(*

.. <legal notes>

legal notes
=================
| SPDX-FileCopyrightText: © 2026 Oleksandr Tiutyk <trofimich@gmail.com>
| SPDX-License-Identifier: LGPL-3.0-only
| For details check: LGPL-3.0-only_

.. _LGPL-3.0-only: https://www.gnu.org/licenses/lgpl-3.0.en.html

.. </legal notes>

*)

TYPE AUTOMATION_CONTROLLER_DIAGNOSTICS :
STRUCT
	InitializationError : AUTOMATION_ERROR_LOG;

	LastEnableError : AUTOMATION_ERROR_LOG;
	LastDisableError : AUTOMATION_ERROR_LOG;
	
	LastSimulationModeChangeError : AUTOMATION_ERROR_LOG;
	
	LastRefreshInputDeviceError : AUTOMATION_ERROR_LOG;
	
	LastRunningError : AUTOMATION_ERROR_LOG;
	LastStoppingError : AUTOMATION_ERROR_LOG;
	LastFaultError : AUTOMATION_ERROR_LOG;
	LastResettingError : AUTOMATION_ERROR_LOG;
	
	LastRefreshOutputDeviceError : AUTOMATION_ERROR_LOG;
	
	LastErrorPalce : STRING(39);
END_STRUCT
END_TYPE

(* stored: Version 1.1.0.1
   DUT AUTOMATION_CONTROLLER_DIAGNOSTICS: Id {bfbf490c-5629-43bf-91fc-3c9a15aee1bf} *)
